// TwinCAT 3 PLC project PLC1
// ProgramVersion: 3.1.4024.0
// libraries:
//   Tc2_ModbusRTU, * (Beckhoff Automation GmbH)
//   Tc2_Standard, * (Beckhoff Automation GmbH)
//   Tc2_System, * (Beckhoff Automation GmbH)
//   Tc3_Module, * (Beckhoff Automation GmbH)
// project tree:
//   DUTs/ E_Modbus_State.TcDUT (not stored), ST_Ecat_State.TcDUT (not stored), U_2Words_toDWord.TcDUT
//   / PlcTask.TcTTO (not stored)
//   POUs/ FB_Ecat_State.TcPOU, FB_Modbus_Rs485.TcPOU, FB_ZA_Fan.TcPOU, MAIN.TcPOU
// real-time tasks:
//   TASK PlcTask: cycle T#10ms, priority 20, ADS port 350
// I/O:
//   DEVICE Device 2 (EtherCAT), AmsNetId 10.33.70.115.3.1
//     Term 1 (EK1100) [EK1100 EtherCAT Coupler (2A E-Bus)] (disabled)
//       Term 2 (EL6021) [EL6021 Interface (RS422/485)]
//       Term 3 (EL6022) [EL6022 Interface 2Ch. (RS422/485)]
//       Term 4 (EL9011) [EL9011 End Terminal]
//     Term 5 (EK1100) [EK1100 EtherCAT Coupler (2A E-Bus)]
//       Term 7 (EL2008) [EL2008 8Ch. Dig. Output 24V, 0.5A]
//       Term 15 (EL6021) [EL6021 Interface (RS422/485)]
//       Term 8 (EL4122) [EL4122 2Ch. Ana. Output  4-20mA, 16bit] (disabled)
//       Term 9 (EL4122) [EL4122 2Ch. Ana. Output  4-20mA, 16bit] (disabled)
//       Term 10 (EL3318) [EL3318 8Ch. Ana Input Thermocouple (TC)] (disabled)
//       Term 11 (EL3318) [EL3318 8Ch. Ana Input Thermocouple (TC)] (disabled)
//       Term 20 (EL6022) [EL6022 Interface 2Ch. (RS422/485)] (disabled)
//       Term 12 (EL9011) [EL9011 End Terminal]
// variable links:
//   PLC1/PLC1 Instance <-> Device 2 (EtherCAT)/Term 5 (EK1100)/Term 15 (EL6021)
//     PlcTask Inputs/MAIN.fbZAFan.fbModbus.fbModbusMaster.InData/D <-> COM TxPDO-Map Inputs/Data In 0
//     PlcTask Inputs/MAIN.fbZAFan.fbModbus.fbModbusMaster.InData/D @bit {8..168 step 8} <-> COM TxPDO-Map Inputs/Data In {1..21}  (21 links)
//     PlcTask Inputs/MAIN.fbZAFan.fbModbus.fbModbusMaster.InData/Status <-> COM TxPDO-Map Inputs/Status
//     PlcTask Inputs/MAIN.fbZAFan.fbModbus.fbModuleEcatState.raw_state/op_state <-> InfoData/State
//     PlcTask Inputs/MAIN.fbZAFan.fbModbus.fbModuleEcatState.raw_state/wc_state <-> WcState/WcState
//     PlcTask Outputs/MAIN.fbZAFan.fbModbus.fbModbusMaster.OutData/Ctrl <-> COM RxPDO-Map Outputs/Ctrl
//     PlcTask Outputs/MAIN.fbZAFan.fbModbus.fbModbusMaster.OutData/D <-> COM RxPDO-Map Outputs/Data Out 0
//     PlcTask Outputs/MAIN.fbZAFan.fbModbus.fbModbusMaster.OutData/D @bit {8..168 step 8} <-> COM RxPDO-Map Outputs/Data Out {1..21}  (21 links)

// ---- DUTs/U_2Words_toDWord.TcDUT
TYPE U_2Words_toDWord :
UNION
	u_words : ARRAY[0..1] OF WORD;
	u_dword : DWORD;
END_UNION
END_TYPE

// ---- POUs/FB_Ecat_State.TcPOU
FUNCTION_BLOCK FB_Ecat_State
VAR_INPUT
END_VAR

VAR
	raw_state AT %I* : ST_Ecat_State;
END_VAR

PROPERTY State : BOOL
GET
State := (NOT raw_state.wc_state) AND raw_state.op_state.3;
END_GET
END_PROPERTY

END_FUNCTION_BLOCK

// ---- POUs/FB_Modbus_Rs485.TcPOU
FUNCTION_BLOCK FB_Modbus_Rs485
VAR_INPUT
	i_slave_id		 	 	: BYTE;
	i_start_read_address 	: WORD;
	i_registers_read_qty			: WORD;	
	i_start_write_address	: WORD;
    i_write_value			: WORD;
END_VAR
	
VAR_OUTPUT
	o_error : BOOL;
	o_commsok : BOOL;
END_VAR

VAR_IN_OUT
	io_raw_data_read			: ARRAY[*] OF WORD;	
	io_write_reg_cmd	: BOOL;
END_VAR

VAR
	fbModuleEcatState : FB_Ecat_State;
	
	fbModbusMaster 														: ModbusRtuMasterV2_KL6x22B;
//	fbModbusMaster 														: ModbusRtuMasterV2_KL6x5B;		
	modbus_state														: E_Modbus_State;
	raw_data_read 														: ARRAY[0..9] OF WORD;
	
	_TIMEOUT_MODBUS														: TIME 		:= T#2S;
	
	size_local_array :  UINT;
	size_io_array : UINT;
	idxReg : DINT;
	error_modbus : BOOL;
	error_id : MODBUS_ERRORS;
	tmrBusy 															: TON;
	sita1																: BOOL;
END_VAR

CASE modbus_state OF
	
	E_Modbus_State.Idle:
		fbModbusMaster(Execute := FALSE);
//		io_write_reg_cmd := FALSE;
		IF NOT o_error AND NOT fbModbusMaster.Error THEN
			modbus_state := E_Modbus_State.ReadInputRegs;
		ELSE
			 modbus_state := E_Modbus_State.Error;
			 o_commsok := FALSE;
		END_IF
		
	
		
	E_Modbus_State.ReadInputRegs:

//		fbModbusMaster.ReadInputRegs(Execute := TRUE);
		
	fbModbusMaster.ReadInputRegs( 
						   Execute 			:= TRUE, 
						   UnitID 			:= i_slave_id,
						   Quantity			:= i_registers_read_qty, 
						   MBAddr			:= i_start_read_address, 
						   cbLength			:= SIZEOF(raw_data_read), 
						   pMemoryAddr		:= ADR(raw_data_read), 				   
						   Timeout			:= _TIMEOUT_MODBUS	);

		IF  NOT fbModbusMaster.BUSY   AND NOT fbModbusMaster.Error THEN
					fbModbusMaster.ReadInputRegs(Execute := FALSE);
					o_commsok := TRUE;
					IF io_write_reg_cmd THEN
						modbus_state := E_Modbus_State.WriteSingleReg;
					END_IF
		ELSIF fbModbusMaster.Error THEN	  
					modbus_state := E_Modbus_State.Error;				
		END_IF	
		
	E_Modbus_State.WriteSingleReg:
		
			
//			fbModbusMaster.WriteSingleRegister(Execute := TRUE);
			fbModbusMaster.WriteSingleRegister(	
							   Execute			:= TRUE,	
							   UnitID 			:= i_slave_id,
							   Quantity			:= 1, 
							   MBAddr			:= i_start_write_address, 
							   cbLength			:= SIZEOF(i_write_value), 
							   pMemoryAddr		:= ADR(i_write_value), 				   
							   Timeout			:= _TIMEOUT_MODBUS	);	
	
			IF  NOT fbModbusMaster.BUSY   AND NOT fbModbusMaster.Error THEN
						fbModbusMaster.WriteSingleRegister(Execute := FALSE);
						io_write_reg_cmd := FALSE;
						modbus_state := E_Modbus_State.ReadInputRegs;
			ELSIF fbModbusMaster.Error THEN	  
						modbus_state := E_Modbus_State.Error;				
			END_IF	
		
		
	E_Modbus_State.Error :
		 o_commsok := FALSE;
		 error_modbus := TRUE;
		 io_write_reg_cmd := FALSE;
		 fbModbusMaster.ReadInputRegs(Execute := FALSE);
		 modbus_state := E_Modbus_State.Error_Reset;
		 
	E_Modbus_State.Error_Reset :
		fbModbusMaster.ReadInputRegs(Execute := TRUE);
		IF NOT fbModbusMaster.BUSY OR NOT fbModbusMaster.Error THEN
			modbus_state := E_Modbus_State.Error_Check;
		END_IF
		
	E_Modbus_State.Error_Check :
	
		IF  NOT fbModbusMaster.Error THEN
//		IF  NOT fbModbusMaster.Error THEN
			error_modbus := FALSE;
			modbus_state := E_Modbus_State.Idle;
		ELSE
			modbus_state := E_Modbus_State.Error;
		END_IF
		
			
	
END_CASE





//fbModbusMaster.ReadInputRegs(  UnitID 			:= i_slave_id,
//							   Quantity			:= i_registers_read_qty, 
//							   MBAddr			:= i_start_read_address, 
//							   cbLength			:= SIZEOF(raw_data_read), 
//							   pMemoryAddr		:= ADR(raw_data_read), 				   
//							   Timeout			:= _TIMEOUT_MODBUS	);
							   

//fbModbusMaster.WriteSingleRegister(	UnitID 			:= i_slave_id,
//							   Quantity			:= 1, 
//							   MBAddr			:= i_start_write_address, 
//							   cbLength			:= SIZEOF(i_write_value), 
//							   pMemoryAddr		:= ADR(i_write_value), 				   
//							   Timeout			:= _TIMEOUT_MODBUS	);				 

					

FOR idxReg := LOWER_BOUND(io_raw_data_read,1) TO UPPER_BOUND(io_raw_data_read,1) DO 
	io_raw_data_read[idxReg] := raw_data_read[idxReg];
END_FOR


o_error  := NOT fbModuleEcatState.State OR error_modbus ;

END_FUNCTION_BLOCK

// ---- POUs/FB_ZA_Fan.TcPOU
FUNCTION_BLOCK FB_ZA_Fan
VAR_INPUT
	i_enable_cmd	: BOOL;
	i_speed_sp		: REAL;
END_VAR
VAR_OUTPUT

END_VAR
VAR
	fbModbus : FB_Modbus_Rs485;
	raw_data_read : ARRAY[0..9] OF WORD;
	modbus_error : BOOL;
	write_cmd : BOOL;
	enable_cmd 	: BOOL;
	speed_sp	: REAL;
	modbus_control_initialized	: BOOL;
	write_address	: WORD;
	write_value		: WORD;
END_VAR

IF modbus_control_initialized AND NOT write_cmd THEN 
	write_value := 0;
	IF i_enable_cmd <> enable_cmd AND NOT write_cmd THEN
		enable_cmd := i_enable_cmd;
		write_address := 1;
		write_value.0 := enable_cmd;
		write_cmd := TRUE;
	END_IF
	IF i_speed_sp <> speed_sp AND NOT write_cmd THEN
		speed_sp := i_speed_sp;
		write_address := 2;
		write_value := TO_WORD(TO_INT(speed_sp));
		write_cmd := TRUE;
	END_IF
END_IF

IF NOT modbus_control_initialized AND NOT write_cmd  AND fbModbus.o_commsok  THEN
	write_value := 0;
	write_address:= 4;
	write_value.0 := TRUE;  //  modbus speed control 
	write_value.9 := TRUE;  // modbus fan enable control 
	write_cmd := TRUE;
	modbus_control_initialized := TRUE;
END_IF


fbModbus(
	i_slave_id:= 247, 
	i_start_read_address:= 1,
	i_registers_read_qty := 5,
	i_start_write_address := write_address, 
	i_write_value := write_value,
	o_error=> modbus_error, 
	io_raw_data_read:= raw_data_read,
	io_write_reg_cmd := write_cmd);

END_FUNCTION_BLOCK

// ---- POUs/MAIN.TcPOU
PROGRAM MAIN
VAR
	
	fbZAFan			 : FB_ZA_Fan;
END_VAR


fbZAFan();

END_PROGRAM
